SUBAPPLICATION SoftKey_Heckschieber_UP (* Subapplication Type *)
  (* Standard: 61499-2 *)
  (* Version 1.0, 2023-02-11, franz *)
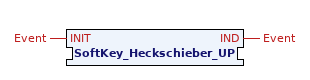
  EVENT_INPUT
    INIT;
  END_EVENT
  EVENT_OUTPUT
    IND;
  END_EVENT
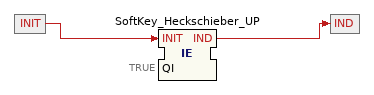
  FBS
    SoftKey_Heckschieber_UP : IE(QI := TRUE);
  END_FBS
  EVENT_CONNECTIONS
    INIT TO SoftKey_Heckschieber_UP.INIT;
    SoftKey_Heckschieber_UP.IND TO IND;
  END_CONNECTIONS
END_SUBAPPLICATION
